TYPE ST_KPI_OutersProduced :
STRUCT
	Total					: UDINT;
	Passed				: UDINT;
	Rejected				: UDINT;
	Efficiency				: LREAL;
END_STRUCT
END_TYPE

(* stored: Version 1.1.0.1
   DUT ST_KPI_OutersProduced: Id {eb33ee2c-e4aa-472b-8ba6-c8c360550f20} *)
